SUBAPPLICATION Uebung_050 (* DigitalInput_I1 auf DigitalOutput_Q1 *)
  (* Standard: 61499-2 *)
  (* Version 1.0, 2023-10-23, franz *)
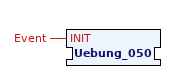
  EVENT_INPUT
    INIT;
  END_EVENT
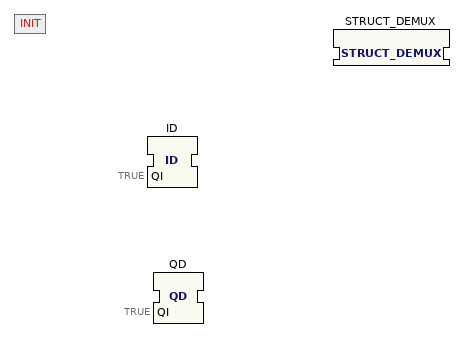
  FBS
    ID : ID(QI := TRUE);
    QD : QD(QI := TRUE);
    STRUCT_DEMUX : STRUCT_DEMUX; {SET_ATTRIBUTE(StructuredType, ANY_STRUCT)}
  END_FBS
END_SUBAPPLICATION
